DATA_BLOCK "RTG1SysInfo"
{InstructionName := 'F_CTRL1';
 LibVersion := '2.2';
 S7_Optimized_Access := 'TRUE' }
AUTHOR : SafeSys
FAMILY : F_CTRL
NAME : F_CTRL_1
VERSION : 2.2
NON_RETAIN
F_CTRL1

BEGIN
   F_SYSINFO.F_PROG_SIG := DW#16#832DEE38;
   F_SYSINFO.F_PROG_DAT := DTL#2021-8-4-22:50:56.862582800;
   F_SYSINFO.F_RTG_SIG := DW#16#F5BD20EF;
   F_SYSINFO.F_RTG_DAT := DTL#2021-8-4-22:50:56.862582800;
   F_SYSINFO.VERS_S7SAF := DW#16#16000000;
   dnMODE_C := 19127;
   dnDB_INIT_C := 70557;
   dnMOD_MODE_C := 34321;
   dnPLCSIM_MODE_C := 20664;
   dnACT_MOD_MODE_C := 27190;
   lnDIFF_C := 35673;
   lnDIFF_MTIME_C := 22975;
   nMAX_CYC := 120;
   dnMAX_CYC_C := 3819182;
   nWARN_CYC := 110;
   dwFCC_VALUE := DW#16#B0695B45;
   dnS_TIM_C := 14080;
   dnS_TIM_ALT_C := 33803;
   dnS_TIM100_CACHE_C := 32709;
   dnS_TIM100_USE_C := 25382;
   dnS_TIM1000_CACHE_C := 26562;
   dnS_TIM1000_USE_C := 41245;
   dnS_DIFF_C := 14080;
   dnS_DIFF100_C := 14080;
   dnS_DIFF1000_C := 14080;
   lnF_TIM_SFC_C := 14080;
   lnF_TIM_SFC_ALT_C := 27889;
   dnF_TIM_C := 14080;
   dnF_TIM_ALT_C := 23998;
   dnF_TIM100_CACHE_C := 26848;
   dnF_TIM100_USE_C := 25044;
   dnF_TIM1000_CACHE_C := 25507;
   dnF_TIM1000_USE_C := 23558;
   dnF_DIFF_C := 14080;
   dnF_DIFF100_C := 14080;
   dnF_DIFF1000_C := 14080;
   dnCONTROL_TIM100_C := 39214;
   dnCONTROL_TIM1000_C := 24463;
   dnTOL_C := 14080;
   dwF_PROG_SIG_DAT_SIG := DW#16#B04411D9;
   dwF_RTG_SIG_DAT_SIG := DW#16#C6D4DF0E;
   wRTG_NO := W#16#1;

END_DATA_BLOCK

